{attribute 'Tc2GvlVarNames'}
{attribute 'strict'}
(* Stato Prodotto GENERICO *)
TYPE e_Stato_Prodotto_Generico :
(
	PROD_ASSENTE	:= 0,	(* Prodotto Assente *)
	PROD_PRESENTE	:= 1	(* Prodotto Presente *)
);
END_TYPE

(* stored: Version 1.1.0.1, ProductVersion 3.1.4024.11
   EnumerationTextList e_Stato_Prodotto_Generico: Id {676e6cbb-309e-4e8b-a035-a4cdad69a2b3} *)
